FUNCTION_BLOCK SimpleDisableWithRotSwAndEstop IMPLEMENTS I_DemoStep
VAR_INPUT
	XPlanarSys	: I_XPlanarSystem;
	M1			: I_XPlanarMover;
	M2			: I_XPlanarMover;
	Track		: I_XPlanarTrack;
	
	SelectorSW	: REFERENCE TO U_SelectorSwitch;
	ESTOP		: REFERENCE TO U_Estop;
END_VAR
VAR_OUTPUT
END_VAR
VAR
	SubStep: USINT;
	_Done: BOOL;
END_VAR

METHOD CyclicLogic
VAR
END_VAR
IF XPlanarSys<>0 AND M1<>0 AND M2<>0 THEN
		//Wait till the mover has completed is current move. Then disable it.
		//That way operator intervention is prevented to re-align the movers, and mover gracefully stops
	IF NOT M1.Status.Busy.busyMover AND NOT M2.Status.Busy.busyMover THEN
		XPlanarSys.DisableMovers();
	END_IF
	_Done:= FALSE;
	IF 	M1.Status.State		= MC_PLANAR_STATE.Disabled 
		AND M2.Status.State	= MC_PLANAR_STATE.Disabled 
		AND (
			( (__ISVALIDREF(SelectorSW) AND __ISVALIDREF(ESTOP) )
				AND_THEN(SelectorSW.Pos = E_SelectorSwitchPos.Left AND Estop.Pos = E_EStop.Normallyclosed) )
		OR XPlanar.OperationMode = XPlanarApplication.XPlanarOperationMode.BasicSimulation)
	THEN
		_Done:= TRUE;
	END_IF
	IF M1.Error THEN
		M1.Reset();
	END_IF

	IF M2.Error THEN
		M2.Reset();
	END_IF
END_IF

IF Track<>0 AND_THEN Track.Error THEN
	Track.Reset();
END_IF
END_METHOD

{attribute 'monitoring' := 'call'}
PROPERTY Done : BOOL
GET
Done:=_Done;
END_GET
END_PROPERTY

METHOD Reset : BOOL
_Done:=FALSE;
SubStep:=0;
Reset:=TRUE;
END_METHOD

END_FUNCTION_BLOCK

(* stored: Version 1.1.0.1, ProductVersion 3.1.4026.21
   POU SimpleDisableWithRotSwAndEstop: Id {e4357684-129c-4ca7-9a46-67b3f6fa6de0}, SpecialFunc None
   Method CyclicLogic: Id {f10e7fd0-de17-4f10-96d9-ef5a94570cfc}
   Property Done: Id {3bedcaca-22b6-48cf-b92b-b5f7072fc0b6}
   Get Get: Id {fc9db926-def4-4b37-8f77-26b4835da4bf}
   Method Reset: Id {21d0da47-9415-4ebd-9bb2-0cfa61d6bd6c} *)
